FUNCTION_BLOCK FB_LogInfoEdge
VAR_INPUT
	Event : BOOL; // Event flag
	Message : T_MaxString; // Log message
	EventFallingEdge : BOOL := FALSE; // Defined which edge: FALSE = rising TRUE = falling, 
END_VAR
VAR_OUTPUT
	Q : BOOL;
END_VAR
VAR
	fbLogEdge : FB_LogOnEdge;
END_VAR

fbLogEdge(
	Event:= Event, 
	Message:= Message, 
	LogSeverity:= E_LogSeverity.Info, 
	EventFallingEdge:= EventFallingEdge,
	Q => Q
);

END_FUNCTION_BLOCK

(* stored: Version 1.1.0.1, ProductVersion 3.1.4020.12
   POU FB_LogInfoEdge: Id {20a97975-5e9f-4e80-b979-474e57877bb0}, SpecialFunc None *)
